// Writes a double field value, without a tag, to the stream.
FUNCTION F_WriteDouble : HRESULT
VAR_INPUT
    stBuffer    : ST_Span;
END_VAR
VAR_IN_OUT
    stState     : ST_WriterInternalState;
END_VAR
VAR_INPUT CONSTANT
    fValue : LREAL;
END_VAR
VAR CONSTANT
    cLength : UDINT := SIZEOF(fValue);
END_VAR
VAR
    fTmp : LREAL;
END_VAR


F_WriteDouble := S_OK;

IF stState.nBufferSize - stState.nBufferPos < cLength THEN
    F_WriteDouble := stState.eWriterErrorCode := E_WriterErrorCode.TruncatedMessage;
    stState.bError := TRUE;
    RETURN;
END_IF
{warning 'TODO: Check for endianess?'}
fTmp := fValue;

MEMCPY(destAddr:= stBuffer.pBuffer + stState.nBufferPos, srcAddr:= ADR(fTmp), n:= cLength);
stState.nBufferPos := stState.nBufferPos + cLength;

END_FUNCTION

(* stored: Version 1.1.0.1
   POU F_WriteDouble: Id {bd6826a6-616d-4379-89c3-33633543bf20}, SpecialFunc None *)
